Universal Robots PolyScope program: Snap_buttom.urp

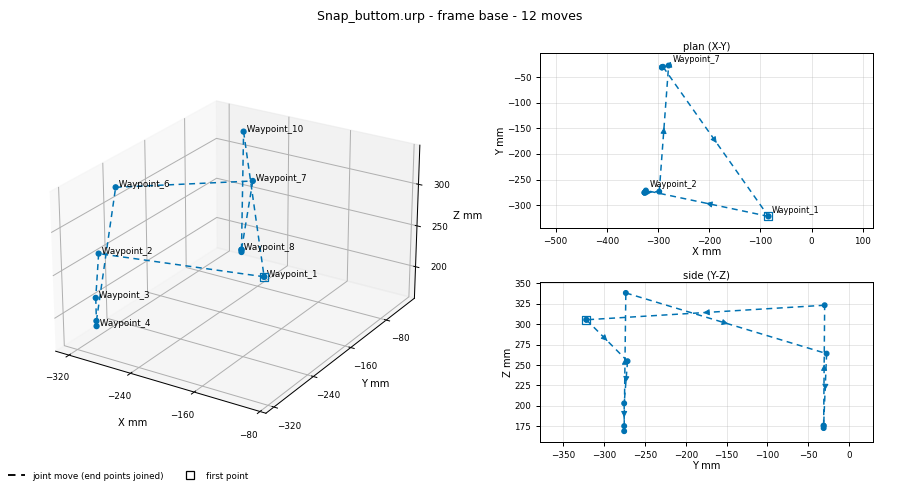
[picture p0: tool path of Snap_buttom.urp in frame base, 12 of 12 moves have a stored position in this frame; points joined in program order, loops and branches not executed]
Program Snap_buttom (installation=default directory=/programs/usbdisk/Zahra1 createdIn=5.11.11.1010533 lastSavedIn=5.11.11.1010533 robotSerialNumber=20205300864)
Calibrated DH parameters: a=[-0.000166, -0.243494, -0.153108, 0.000057, -0.000123, 0]; d=[0.151897, -1.34267, 53.988124, -52.514559, 0.085283, 0.092193]; alpha=[1.572472, -0.003756, 0.002824, 1.570807, -1.572621, 0]; deltaTheta=[0, 0.020704, 7.033215, -0.770746, 0.000004, 0]
Robot Program (runOnlyOnce=true)
  MoveJ speed 60 deg/s, acceleration 80 deg/s^2 (useActiveTCP=true) feature=Base
    Waypoint Waypoint_1: TCP in base x=-84.299 y=-321.875 z=305.481 mm, rx=-2.0809 ry=-2.2572 rz=0.0984 rad; joints [-79.978, -91.201, -87.971, -91.7, 84.671, 815.506] deg
    URCap Gripper (Robotiq_Grippers, Robotiq Inc.) dataModel(position=33.72549019607843, force=94.0, speed=40.0, positionInDouble=33.72549019607843, forceInDouble=94.0, speedInDouble=40.0, slaveIds=[9], blocking=true, robotCompliant=false)
    Waypoint Waypoint_2: TCP in base x=-323.667 y=-271.393 z=254.671 mm, rx=-2.193 ry=-2.2427 rz=0.0752 rad; joints [-121.855, -114.418, -73.91, -78.935, 89.127, 776.94] deg
    Waypoint Waypoint_3: TCP in base x=-326.224 y=-275.524 z=202.96 mm, rx=2.1997 ry=2.2313 rz=-0.0431 rad; joints [-122.083, -118.968, -80.862, -68.425, 90.056, 777.225] deg
    Waypoint Waypoint_4: TCP in base x=-326.238 y=-275.529 z=168.816 mm, rx=2.1997 ry=2.2311 rz=-0.0433 rad; joints [-122.098, -122.234, -85.549, -60.463, 90.057, 777.228] deg
    URCap Gripper (Robotiq_Grippers, Robotiq Inc.) dataModel(position=62.431372549019606, force=94.0, speed=40.0, positionInDouble=62.431372549019606, forceInDouble=94.0, speedInDouble=40.0, slaveIds=[9], blocking=true, robotCompliant=false)
    Waypoint Waypoint_5: TCP in base x=-326.234 y=-275.522 z=175.099 mm, rx=2.1996 ry=2.2312 rz=-0.0431 rad; joints [-122.096, -121.559, -84.785, -61.91, 90.059, 777.225] deg
    Waypoint Waypoint_6: TCP in base x=-297.554 y=-273.504 z=338.378 mm, rx=-2.2095 ry=-2.19 rz=0.0516 rad; joints [-118.013, -110.705, -56.075, -101.815, 87.698, 782.531] deg
    Waypoint Waypoint_7: TCP in base x=-279.278 y=-27.274 z=263.977 mm, rx=2.1983 ry=2.2417 rz=-0.0702 rad; joints [-146.962, -78.086, -112.234, -77.086, 90.697, 752.056] deg
    Waypoint Waypoint_8: TCP in base x=-292.327 y=-30.901 z=175.586 mm, rx=-2.228 ry=-2.2046 rz=-0.0067 rad; joints [-147.51, -91.612, -125.138, -53.3, 89.609, 753.289] deg
    Waypoint Waypoint_9: TCP in base x=-292.342 y=-30.891 z=172.644 mm, rx=-2.228 ry=-2.2046 rz=-0.0067 rad; joints [-147.514, -92.127, -125.591, -52.329, 89.605, 753.29] deg
    URCap Gripper (Robotiq_Grippers, Robotiq Inc.) dataModel(position=25.098039215686274, force=94.0, speed=40.0, positionInDouble=25.098039215686274, forceInDouble=94.0, speedInDouble=40.0, slaveIds=[9], blocking=true, robotCompliant=false)
    Waypoint Waypoint_8: TCP in base x=-292.327 y=-30.901 z=175.586 mm, rx=-2.228 ry=-2.2046 rz=-0.0067 rad; joints [-147.51, -91.612, -125.138, -53.3, 89.609, 753.289] deg
    Waypoint Waypoint_10: TCP in base x=-290.336 y=-29.667 z=323.298 mm, rx=-2.2522 ry=-2.1784 rz=0.008 rad; joints [-147.467, -81.148, -92.919, -95.447, 89.642, 754.53] deg
    Waypoint Waypoint_1: TCP in base x=-84.299 y=-321.875 z=305.481 mm, rx=-2.0809 ry=-2.2572 rz=0.0984 rad; joints [-79.978, -91.201, -87.971, -91.7, 84.671, 815.506] deg
